TEST_FINISHED();
END_METHOD

METHOD PRIVATE Test_SINT
VAR
    a : SINT := 100;
    result : U_ExpectedOrActual;
END_VAR
TEST('Test_SINT');

result := TcUnit.F_AnyToUnionValue(AnyValue := a);

AssertEquals(Expected := a,
             Actual := result.sintExpectedOrActual,
             Message := 'Values differ');

TEST_FINISHED();
END_METHOD

METHOD PRIVATE Test_STRING
VAR
    a : STRING := 'This is a random string';
    result : U_ExpectedOrActual;
END_VAR
TEST('Test_STRING');

result := TcUnit.F_AnyToUnionValue(AnyValue := a);

AssertEquals(Expected := a,
             Actual := result.stringExpectedOrActual,
             Message := 'Values differ');

TEST_FINISHED();
END_METHOD

METHOD PRIVATE Test_STRING_2
VAR
    a : Tc2_System.T_MaxString := '8YNn5KOmPC4dAcpOBdLWnw4WkN126EwXsj65xeurG48gWBepinNaOIKeCVMtWNBSxQWPdtUYiAusDkjMLtQhDtiWbwvmoKcFwiUGDd7pOe0fd52J7hK60oaYAX6VWWmceLJX8utaDVrVzCGXafeZLeHl6jj5enfjg4tfb2WMEBdsBuG2iDKwzwhBLCPqXDnhe5HbemIbtZT7p62OEj2oDqiIYDD6tZdlhBCCelDBx6dbIp32wFm0TpRKsTiwkZ6'; // 255 characters
    result : U_ExpectedOrActual;
END_VAR
TEST('Test_STRING_2');

result := TcUnit.F_AnyToUnionValue(AnyValue := a);

AssertEquals(Expected := a,
             Actual := result.stringExpectedOrActual,
             Message := 'Values differ');

TEST_FINISHED();
END_METHOD

METHOD PRIVATE Test_TIME
VAR
    a : TIME := T#15M20S;
    result : U_ExpectedOrActual;
END_VAR
TEST('Test_TIME');

result := TcUnit.F_AnyToUnionValue(AnyValue := a);

AssertEquals(Expected := a,
             Actual := result.timeExpectedOrActual,
             Message := 'Values differ');

TEST_FINISHED();
END_METHOD

METHOD PRIVATE Test_TIME_OF_DAY
VAR
    a : TIME_OF_DAY := TOD#15:36:30.123;
    result : U_ExpectedOrActual;
END_VAR
TEST('Test_TIME_OF_DAY');

result := TcUnit.F_AnyToUnionValue(AnyValue := a);

AssertEquals(Expected := a,
             Actual := result.timeofdayExpectedOrActual,
             Message := 'Values differ');

TEST_FINISHED();
END_METHOD

METHOD PRIVATE Test_UDINT
VAR
    a : UDINT := 2555;
    result : U_ExpectedOrActual;
END_VAR
TEST('Test_UDINT');

result := TcUnit.F_AnyToUnionValue(AnyValue := a);

AssertEquals(Expected := a,
             Actual := result.udintExpectedOrActual,
             Message := 'Values differ');

TEST_FINISHED();
END_METHOD

METHOD PRIVATE Test_UINT
VAR
    a : UINT := 34523;
    result : U_ExpectedOrActual;
END_VAR
TEST('Test_UINT');

result := TcUnit.F_AnyToUnionValue(AnyValue := a);

AssertEquals(Expected := a,
             Actual := result.uintExpectedOrActual,
             Message := 'Values differ');

TEST_FINISHED();
END_METHOD

METHOD PRIVATE Test_ULINT
VAR
    a : ULINT := 25555423;
    result : U_ExpectedOrActual;
END_VAR
TEST('TEST_ULINT');

result := TcUnit.F_AnyToUnionValue(AnyValue := a);

AssertEquals(Expected := a,
             Actual := result.ulintExpectedOrActual,
             Message := 'Values differ');

TEST_FINISHED();
END_METHOD

METHOD PRIVATE Test_USINT
VAR
    a : USINT := 255;
    result : U_ExpectedOrActual;
END_VAR
TEST('Test_USINT');

result := TcUnit.F_AnyToUnionValue(AnyValue := a);

AssertEquals(Expected := a,
             Actual := result.usintExpectedOrActual,
             Message := 'Values differ');

TEST_FINISHED();
END_METHOD

METHOD PRIVATE Test_WORD
VAR
    a : WORD := 16#ABCD;
    result : U_ExpectedOrActual;
END_VAR
TEST('Test_WORD');

result := TcUnit.F_AnyToUnionValue(AnyValue := a);

AssertEquals(Expected := a,
             Actual := result.wordExpectedOrActual,
             Message := 'Values differ');

TEST_FINISHED();
END_METHOD

METHOD PRIVATE Test_WSTRING
VAR
    a : WSTRING := "This is a random string";
    result : U_ExpectedOrActual;
END_VAR
TEST('Test_WSTRING');

result := TcUnit.F_AnyToUnionValue(AnyValue := a);

AssertEquals(Expected := a,
             Actual := result.wstringExpectedOrActual,
             Message := 'Values differ');

TEST_FINISHED();
END_METHOD

END_FUNCTION_BLOCK

// ---- Test/FB_MultipleAssertWithSameParametersInSameCycleWithSameTest.TcPOU
(*
    This test-suite runs several asserts with the same parameters (same expected, actual, message) in the same cycle
    and in the same test.
    The reason we want the framework to support this is that theoretically the user could want to do an assert with the
    same message, in the same test, with the same data values for both expected and actual, although the data that the
    user does the assert on might be from different data sets.
*)
FUNCTION_BLOCK FB_MultipleAssertWithSameParametersInSameCycleWithSameTest EXTENDS TcUnit.FB_TestSuite

Assert_SeveralTimes();

METHOD PRIVATE Assert_SeveralTimes
VAR
    a : DWORD := 16#12345678;
    b : DWORD := 16#90ABCDEF;

    c : DWORD := 16#12345678;
    d : DWORD := 16#90ABCDEF;

    e : DWORD := 16#12345678;
    f : DWORD := 16#90ABCDEF;
END_VAR
TEST('Assert_SeveralTimes');

AssertEquals_DWORD(Expected := a,
                   Actual := b,
                   Message := 'Values differ');

AssertEquals_DWORD(Expected := c,
                   Actual := d,
                   Message := 'Values differ');

AssertEquals_DWORD(Expected := e,
                   Actual := f,
                   Message := 'Values differ');

TEST_FINISHED();
END_METHOD

END_FUNCTION_BLOCK

// ---- Test/FB_MultipleAssertWithSameParametersInDifferentCyclesButWithDifferentTests.TcPOU
(*
    This test-suite runs several asserts with the same parameters (same expected, actual, message), calling the asserts
    in different cycles and using different tests.
    On top of this, we will call new asserts (though with same parameters) in later cycles.
    The reason we want the framework to support this is that theoretically the user could want to do an assert with the
    same message, in different tests, with the same data values for both expected and actual, although the data that the
    user does the assert on might be from different data sets.
*)
{attribute 'call_after_init'}
FUNCTION_BLOCK FB_MultipleAssertWithSameParametersInDifferentCyclesButWithDifferentTests EXTENDS TcUnit.FB_TestSuite
VAR
    TimerAgain : Tc2_Standard.TON := (PT := T#1S); // Timer to call "AssertSeveralTimesAgain"
    TimerAgainAgain : Tc2_Standard.TON := (PT := T#5S); // Timer to call "AssertSeveralTimesAgainAgain"
    CalledAll : BOOL; // Indication of whether we've called all tests
END_VAR

TimerAgain(IN := TRUE);

Assert_SeveralTimes();

IF TimerAgain.Q THEN
    TimerAgainAgain(IN := TRUE);
    Assert_SeveralTimesAgain();
END_IF

IF TimerAgainAgain.Q THEN
    Assert_SeveralTimesAgainAgain();
    CalledAll := TRUE;
END_IF

METHOD PRIVATE Assert_SeveralTimes
VAR
    a : DWORD := 16#12345678;
    b : DWORD := 16#90ABCDEF;

    c : DWORD := 16#12345678;
    d : DWORD := 16#90ABCDEF;

    e : DWORD := 16#12345678;
    f : DWORD := 16#90ABCDEF;
END_VAR
TEST('Assert_SeveralTimes');

AssertEquals_DWORD(Expected := a,
                   Actual := b,
                   Message := 'Values differ');

AssertEquals_DWORD(Expected := c,
                   Actual := d,
                   Message := 'Values differ');

AssertEquals_DWORD(Expected := e,
                   Actual := f,
                   Message := 'Values differ');

IF CalledAll THEN
    TEST_FINISHED();
END_IF
END_METHOD

METHOD PRIVATE Assert_SeveralTimesAgain
VAR
    a : DWORD := 16#12345678;
    b : DWORD := 16#90ABCDEF;

    c : DWORD := 16#12345678;
    d : DWORD := 16#90ABCDEF;

    e : DWORD := 16#12345678;
    f : DWORD := 16#90ABCDEF;
END_VAR
TEST('Assert_SeveralTimesAgain');

AssertEquals_DWORD(Expected := a,
                   Actual := b,
                   Message := 'Values differ');

AssertEquals_DWORD(Expected := c,
                   Actual := d,
                   Message := 'Values differ');

AssertEquals_DWORD(Expected := e,
                   Actual := f,
                   Message := 'Values differ');

IF CalledAll THEN
    TEST_FINISHED();
END_IF
END_METHOD

METHOD PRIVATE Assert_SeveralTimesAgainAgain
VAR
    a : DWORD := 16#12345678;
    b : DWORD := 16#90ABCDEF;

    c : DWORD := 16#12345678;
    d : DWORD := 16#90ABCDEF;

    e : DWORD := 16#12345678;
    f : DWORD := 16#90ABCDEF;
END_VAR
TEST('Assert_SeveralTimesAgainAgain');

AssertEquals_DWORD(Expected := a,
                   Actual := b,
                   Message := 'Values differ');

AssertEquals_DWORD(Expected := c,
                   Actual := d,
                   Message := 'Values differ');

AssertEquals_DWORD(Expected := e,
                   Actual := f,
                   Message := 'Values differ');

IF CalledAll THEN
    TEST_FINISHED();
END_IF
END_METHOD

END_FUNCTION_BLOCK

// ---- Test/FB_MultipleAssertWithSameParametersInDifferentCyclesAndInSameTest.TcPOU
(*
    This test-suite runs several asserts with the same parameters (same expected, actual, message), calling the asserts
    in different cycles and using the same test.
    On top of this, we will call new asserts (though with same parameters) in later cycles.
    The reason we want the framework to support this is that theoretically the user could want to do an assert with the
    same message, using the same test with the same data values for both expected and actual, and splitting the asserts
    on different cycles.
*)
FUNCTION_BLOCK FB_MultipleAssertWithSameParametersInDifferentCyclesAndInSameTest EXTENDS TcUnit.FB_TestSuite
VAR
    TimerAgain : Tc2_Standard.TON := (PT := T#1S); // Timer to call "AssertSeveralTimesAgain"
    TimerAgainAgain : Tc2_Standard.TON := (PT := T#5S); // Timer to call "AssertSeveralTimesAgainAgain"
    CalledAll : BOOL; // Indication of whether we've called all tests
END_VAR

Assert_SeveralTimes();

METHOD PRIVATE Assert_SeveralTimes
VAR
    a : DWORD := 16#12345678;
    b : DWORD := 16#90ABCDEF;

    c : DWORD := 16#12345678;
    d : DWORD := 16#90ABCDEF;

    e : DWORD := 16#12345678;
    f : DWORD := 16#90ABCDEF;

    g : DWORD := 16#12345678;
    h : DWORD := 16#90ABCDEF;

    i : DWORD := 16#12345678;
    j : DWORD := 16#90ABCDEF;

    k : DWORD := 16#12345678;
    l : DWORD := 16#90ABCDEF;

    m : DWORD := 16#12345678;
    n : DWORD := 16#90ABCDEF;

    o : DWORD := 16#12345678;
    p : DWORD := 16#90ABCDEF;

    q : DWORD := 16#12345678;
    rr : DWORD := 16#90ABCDEF;
END_VAR
TEST('Assert_SeveralTimes');

AssertEquals_DWORD(Expected := a,
                   Actual := b,
                   Message := 'Values differ');
AssertEquals_DWORD(Expected := c,
                   Actual := d,
                   Message := 'Values differ');
AssertEquals_DWORD(Expected := e,
                   Actual := f,
                   Message := 'Values differ');

TimerAgain(IN := TRUE);
IF TimerAgain.Q THEN
    TimerAgainAgain(IN := TRUE);
    AssertEquals_DWORD(Expected := g,
                       Actual := h,
                       Message := 'Values differ');
    AssertEquals_DWORD(Expected := i,
                       Actual := j,
                       Message := 'Values differ');
    AssertEquals_DWORD(Expected := k,
                       Actual := l,
                       Message := 'Values differ');
END_IF

IF TimerAgainAgain.Q THEN
    AssertEquals_DWORD(Expected := m,
                       Actual := n,
                       Message := 'Values differ');
    AssertEquals_DWORD(Expected := o,
                       Actual := p,
                       Message := 'Values differ');
    AssertEquals_DWORD(Expected := q,
                       Actual := rr,
                       Message := 'Values differ');
    CalledAll := TRUE;
    TEST_FINISHED();
END_IF
END_METHOD

END_FUNCTION_BLOCK

// ---- Test/FB_SkipAssertionsWhenFinished.TcPOU
(*
    Contains tests that require multiple cycles:
    - A short test that finishes quickly
        - The assert statements all pass while the test is not finished
        - After the test is finished, the variables change so that the assert statements now fail,
            which shouldn't matter because the test is finished
    - A long test that finishes slowly
        - This test exists so that the entire test suite keeps running after the short test finishes
*)
FUNCTION_BLOCK FB_SkipAssertionsWhenFinished EXTENDS TcUnit.FB_TestSuite
VAR
    ShortTimer : Tc2_Standard.TON := (PT := T#200MS);
    LongTimer : Tc2_Standard.TON := (PT := T#1S);
END_VAR

Test_LongTest(ADR(LongTimer));
Test_ShortTest(ADR(ShortTimer));
Test_AssertImmediatelyAfterFinished();

(*
    Assertions called immediately after (and within the same cycle as) TEST_FINISHED should be
    ignored.
*)
METHOD Test_AssertImmediatelyAfterFinished
TEST('Test_AssertImmediatelyAfterFinished');
TEST_FINISHED();

AssertTrue(FALSE, 'This failing assertion should be skipped because the test is finished');
END_METHOD

METHOD Test_LongTest
VAR_INPUT
    Timer : POINTER TO Tc2_Standard.TON;
END_VAR
TEST('Test_LongTest');

Timer^(IN := TRUE);
IF Timer^.Q THEN
    TEST_FINISHED();
END_IF
END_METHOD

METHOD Test_ShortTest
VAR_INPUT
    Timer : POINTER TO Tc2_Standard.TON;
END_VAR
TEST('Test_ShortTest');

AssertFalse(Timer^.Q, 'This assertion will start to fail after the test is over, but it will be skipped at that point');

Timer^(IN := TRUE);
IF Timer^.Q THEN
    TEST_FINISHED();
END_IF
END_METHOD

END_FUNCTION_BLOCK

// ---- Test/FB_EmptyTestSuite.TcPOU
(* This is an empty testsuite with no test cases, so that we can verify that the system still prints the
   test results. *)
FUNCTION_BLOCK FB_EmptyTestSuite EXTENDS TcUnit.FB_TestSuite
VAR
END_VAR

END_FUNCTION_BLOCK

// ---- Test/FB_CheckIfSpecificTestIsFinished.TcPOU
(*
    Verifies that the function IS_TEST_FINISHED('Name') works as intended.
*)
FUNCTION_BLOCK FB_CheckIfSpecificTestIsFinished EXTENDS TcUnit.FB_TestSuite

CheckBeforeAndAfterFinishing();

METHOD CheckBeforeAndAfterFinishing
TEST('CheckBeforeAndAfterFinishing');

AssertEquals_BOOL(Expected := FALSE,
                  Actual := IS_TEST_FINISHED('CheckBeforeAndAfterFinishing'),
                  Message:='Values differ before finishing');

TEST_FINISHED();

AssertEquals_BOOL(Expected := TRUE,
                  Actual := IS_TEST_FINISHED('CheckBeforeAndAfterFinishing'),
                  Message:='Values differ after finishing');
END_METHOD

END_FUNCTION_BLOCK

// ---- Test/FB_WriteProtectedFunctions.TcPOU
(*
    This testsuite tests the WRITE_PROTECTED_* helper functions.
*)
FUNCTION_BLOCK FB_WriteProtectedFunctions EXTENDS TcUnit.FB_TestSuite

Test_WRITE_PROTECTED_BOOL();
Test_WRITE_PROTECTED_BYTE();
Test_WRITE_PROTECTED_DATE();
Test_WRITE_PROTECTED_DATE_AND_TIME();
Test_WRITE_PROTECTED_DINT();
Test_WRITE_PROTECTED_DWORD();
Test_WRITE_PROTECTED_INT();
Test_WRITE_PROTECTED_LREAL();
Test_WRITE_PROTECTED_REAL();
Test_WRITE_PROTECTED_SINT();
Test_WRITE_PROTECTED_STRING();
Test_WRITE_PROTECTED_TIME();
Test_WRITE_PROTECTED_TIME_OF_DAY();
Test_WRITE_PROTECTED_UDINT();
Test_WRITE_PROTECTED_UINT();
Test_WRITE_PROTECTED_USINT();
Test_WRITE_PROTECTED_WORD();

METHOD Test_WRITE_PROTECTED_BOOL
VAR
    ProtectedVariables : FB_ProtectedVariables;
END_VAR
TEST('Test_WRITE_PROTECTED_BOOL');

WRITE_PROTECTED_BOOL(ADR(ProtectedVariables.InputBOOL), TRUE);
AssertEquals_BOOL(TRUE, ProtectedVariables.InputBOOL, 'Overwriting protected InputBOOL');

WRITE_PROTECTED_BOOL(ADR(ProtectedVariables.VarBOOL), TRUE);
AssertEquals_BOOL(TRUE, ProtectedVariables.VarBOOL, 'Overwriting protected VarBOOL');

TEST_FINISHED();
END_METHOD

METHOD Test_WRITE_PROTECTED_BYTE
VAR
    ProtectedVariables : FB_ProtectedVariables;
END_VAR
TEST('Test_WRITE_PROTECTED_BYTE');

WRITE_PROTECTED_BYTE(ADR(ProtectedVariables.InputBYTE), 1);
AssertEquals_BYTE(1, ProtectedVariables.InputBYTE, 'Overwriting protected InputBYTE');

WRITE_PROTECTED_BYTE(ADR(ProtectedVariables.VarBYTE), 1);
AssertEquals_BYTE(1, ProtectedVariables.VarBYTE, 'Overwriting protected VarBYTE');

TEST_FINISHED();
END_METHOD

METHOD Test_WRITE_PROTECTED_DATE
VAR
    ProtectedVariables : FB_ProtectedVariables;
END_VAR
TEST('Test_WRITE_PROTECTED_DATE');

WRITE_PROTECTED_DATE(ADR(ProtectedVariables.InputDATE), D#2000-01-01);
AssertEquals_DATE(D#2000-01-01, ProtectedVariables.InputDATE, 'Overwriting protected InputDATE');

WRITE_PROTECTED_DATE(ADR(ProtectedVariables.VarDATE), D#2000-01-01);
AssertEquals_DATE(D#2000-01-01, ProtectedVariables.VarDATE, 'Overwriting protected VarDATE');

TEST_FINISHED();
END_METHOD

METHOD Test_WRITE_PROTECTED_DATE_AND_TIME
VAR
    ProtectedVariables : FB_ProtectedVariables;
END_VAR
TEST('Test_WRITE_PROTECTED_DATE_AND_TIME');

WRITE_PROTECTED_DATE_AND_TIME(ADR(ProtectedVariables.InputDATE_AND_TIME), DT#2000-01-01-00:00);
AssertEquals_DATE_AND_TIME(DT#2000-01-01-00:00, ProtectedVariables.InputDATE_AND_TIME, 'Overwriting protected InputDATE_AND_TIME');

WRITE_PROTECTED_DATE_AND_TIME(ADR(ProtectedVariables.VarDATE_AND_TIME), DT#2000-01-01-00:00);
AssertEquals_DATE_AND_TIME(DT#2000-01-01-00:00, ProtectedVariables.VarDATE_AND_TIME, 'Overwriting protected VarDATE_AND_TIME');

TEST_FINISHED();
END_METHOD

METHOD Test_WRITE_PROTECTED_DINT
VAR
    ProtectedVariables : FB_ProtectedVariables;
END_VAR
TEST('Test_WRITE_PROTECTED_DINT');

WRITE_PROTECTED_DINT(ADR(ProtectedVariables.InputDINT), 1);
AssertEquals_DINT(1, ProtectedVariables.InputDINT, 'Overwriting protected InputDINT');

WRITE_PROTECTED_DINT(ADR(ProtectedVariables.VarDINT), 1);
AssertEquals_DINT(1, ProtectedVariables.VarDINT, 'Overwriting protected VarDINT');

TEST_FINISHED();
END_METHOD

METHOD Test_WRITE_PROTECTED_DWORD
VAR
    ProtectedVariables : FB_ProtectedVariables;
END_VAR
TEST('Test_WRITE_PROTECTED_DWORD');

WRITE_PROTECTED_DWORD(ADR(ProtectedVariables.InputDWORD), 1);
AssertEquals_DWORD(1, ProtectedVariables.InputDWORD, 'Overwriting protected InputDWORD');

WRITE_PROTECTED_DWORD(ADR(ProtectedVariables.VarDWORD), 1);
AssertEquals_DWORD(1, ProtectedVariables.VarDWORD, 'Overwriting protected VarDWORD');

TEST_FINISHED();
END_METHOD

METHOD Test_WRITE_PROTECTED_INT
VAR
    ProtectedVariables : FB_ProtectedVariables;
END_VAR
TEST('Test_WRITE_PROTECTED_INT');

WRITE_PROTECTED_INT(ADR(ProtectedVariables.InputINT), 1);
AssertEquals_INT(1, ProtectedVariables.InputINT, 'Overwriting protected InputINT');

WRITE_PROTECTED_INT(ADR(ProtectedVariables.VarINT), 1);
AssertEquals_INT(1, ProtectedVariables.VarINT, 'Overwriting protected VarINT');

TEST_FINISHED();
END_METHOD

METHOD Test_WRITE_PROTECTED_LREAL
VAR
    ProtectedVariables : FB_ProtectedVariables;
END_VAR
TEST('Test_WRITE_PROTECTED_LREAL');

WRITE_PROTECTED_LREAL(ADR(ProtectedVariables.InputLREAL), 1);
AssertEquals_LREAL(1, ProtectedVariables.InputLREAL, 0, 'Overwriting protected InputLREAL');

WRITE_PROTECTED_LREAL(ADR(ProtectedVariables.VarLREAL), 1);
AssertEquals_LREAL(1, ProtectedVariables.VarLREAL, 0, 'Overwriting protected VarLREAL');

TEST_FINISHED();
END_METHOD

METHOD Test_WRITE_PROTECTED_REAL
VAR
    ProtectedVariables : FB_ProtectedVariables;
END_VAR
TEST('Test_WRITE_PROTECTED_REAL');

WRITE_PROTECTED_REAL(ADR(ProtectedVariables.InputREAL), 1);
AssertEquals_REAL(1, ProtectedVariables.InputREAL, 0, 'Overwriting protected InputREAL');

WRITE_PROTECTED_REAL(ADR(ProtectedVariables.VarREAL), 1);
AssertEquals_REAL(1, ProtectedVariables.VarREAL, 0, 'Overwriting protected VarREAL');

TEST_FINISHED();
END_METHOD

METHOD Test_WRITE_PROTECTED_SINT
VAR
    ProtectedVariables : FB_ProtectedVariables;
END_VAR
TEST('Test_WRITE_PROTECTED_SINT');

WRITE_PROTECTED_SINT(ADR(ProtectedVariables.InputSINT), 1);
AssertEquals_SINT(1, ProtectedVariables.InputSINT, 'Overwriting protected InputSINT');

WRITE_PROTECTED_SINT(ADR(ProtectedVariables.VarSINT), 1);
AssertEquals_SINT(1, ProtectedVariables.VarSINT, 'Overwriting protected VarSINT');

TEST_FINISHED();
END_METHOD

METHOD Test_WRITE_PROTECTED_STRING
VAR
    ProtectedVariables : FB_ProtectedVariables;
END_VAR
TEST('Test_WRITE_PROTECTED_STRING');

WRITE_PROTECTED_STRING(ADR(ProtectedVariables.InputSTRING), 'words');
AssertEquals_STRING('words', ProtectedVariables.InputSTRING, 'Overwriting protected InputSTRING');

WRITE_PROTECTED_STRING(ADR(ProtectedVariables.VarSTRING), 'words');
AssertEquals_STRING('words', ProtectedVariables.VarSTRING, 'Overwriting protected VarSTRING');

TEST_FINISHED();
END_METHOD

METHOD Test_WRITE_PROTECTED_TIME
VAR
    ProtectedVariables : FB_ProtectedVariables;
END_VAR
TEST('Test_WRITE_PROTECTED_TIME');

WRITE_PROTECTED_TIME(ADR(ProtectedVariables.InputTIME), T#1S);
AssertEquals_TIME(T#1S, ProtectedVariables.InputTIME, 'Overwriting protected InputTIME');

WRITE_PROTECTED_TIME(ADR(ProtectedVariables.VarTIME), T#1S);
AssertEquals_TIME(T#1S, ProtectedVariables.VarTIME, 'Overwriting protected VarTIME');

TEST_FINISHED();
END_METHOD

METHOD Test_WRITE_PROTECTED_TIME_OF_DAY
VAR
    ProtectedVariables : FB_ProtectedVariables;
END_VAR
TEST('Test_WRITE_PROTECTED_TIME_OF_DAY');

WRITE_PROTECTED_TIME_OF_DAY(ADR(ProtectedVariables.InputTIME_OF_DAY), TOD#11:11);
AssertEquals_TIME_OF_DAY(TOD#11:11, ProtectedVariables.InputTIME_OF_DAY, 'Overwriting protected InputTIME_OF_DAY');

WRITE_PROTECTED_TIME_OF_DAY(ADR(ProtectedVariables.VarTIME_OF_DAY), TOD#11:11);
AssertEquals_TIME_OF_DAY(TOD#11:11, ProtectedVariables.VarTIME_OF_DAY, 'Overwriting protected VarTIME_OF_DAY');

TEST_FINISHED();
END_METHOD

METHOD Test_WRITE_PROTECTED_UDINT
VAR
    ProtectedVariables : FB_ProtectedVariables;
END_VAR
TEST('Test_WRITE_PROTECTED_UDINT');

WRITE_PROTECTED_UDINT(ADR(ProtectedVariables.InputUDINT), 1);
AssertEquals_UDINT(1, ProtectedVariables.InputUDINT, 'Overwriting protected InputUDINT');

WRITE_PROTECTED_UDINT(ADR(ProtectedVariables.VarUDINT), 1);
AssertEquals_UDINT(1, ProtectedVariables.VarUDINT, 'Overwriting protected VarUDINT');

TEST_FINISHED();
END_METHOD

METHOD Test_WRITE_PROTECTED_UINT
VAR
    ProtectedVariables : FB_ProtectedVariables;
END_VAR
TEST('Test_WRITE_PROTECTED_UINT');

WRITE_PROTECTED_UINT(ADR(ProtectedVariables.InputUINT), 1);
AssertEquals_UINT(1, ProtectedVariables.InputUINT, 'Overwriting protected InputUINT');

WRITE_PROTECTED_UINT(ADR(ProtectedVariables.VarUINT), 1);
AssertEquals_UINT(1, ProtectedVariables.VarUINT, 'Overwriting protected VarUINT');

TEST_FINISHED();
END_METHOD

METHOD Test_WRITE_PROTECTED_USINT
VAR
    ProtectedVariables : FB_ProtectedVariables;
END_VAR
TEST('Test_WRITE_PROTECTED_USINT');

WRITE_PROTECTED_USINT(ADR(ProtectedVariables.InputUSINT), 1);
AssertEquals_USINT(1, ProtectedVariables.InputUSINT, 'Overwriting protected InputUSINT');

WRITE_PROTECTED_USINT(ADR(ProtectedVariables.VarUSINT), 1);
AssertEquals_USINT(1, ProtectedVariables.VarUSINT, 'Overwriting protected VarUSINT');

TEST_FINISHED();
END_METHOD

METHOD Test_WRITE_PROTECTED_WORD
VAR
    ProtectedVariables : FB_ProtectedVariables;
END_VAR
TEST('Test_WRITE_PROTECTED_WORD');

WRITE_PROTECTED_WORD(ADR(ProtectedVariables.InputWORD), 1);
AssertEquals_WORD(1, ProtectedVariables.InputWORD, 'Overwriting protected InputWORD');

WRITE_PROTECTED_WORD(ADR(ProtectedVariables.VarWORD), 1);
AssertEquals_WORD(1, ProtectedVariables.VarWORD, 'Overwriting protected VarWORD');

TEST_FINISHED();
END_METHOD

END_FUNCTION_BLOCK

// ---- POUs/FB_ProtectedVariables.TcPOU
(*
    Contains different types of "protected" variables that you could not normally write to in
    production PLC code, but would need to overwrite for testing purposes. Used for testing the
    WRITE_PROTECTED_* functions, but this FB doesn't contain any tests itself.
*)
FUNCTION_BLOCK FB_ProtectedVariables
VAR_INPUT
    InputBOOL AT %I* : BOOL;
    InputBYTE AT %I* : BYTE;
    InputDATE AT %I* : DATE;
    InputDATE_AND_TIME AT %I* : DATE_AND_TIME;
    InputDINT AT %I* : DINT;
    InputDWORD AT %I* : DWORD;
    InputINT AT %I* : INT;
    InputLREAL AT %I* : LREAL;
    InputREAL AT %I* : REAL;
    InputSINT AT %I* : SINT;
    InputSTRING AT %I* : STRING;
    InputTIME AT %I* : TIME;
    InputTIME_OF_DAY AT %I* : TIME_OF_DAY;
    InputUDINT AT %I* : UDINT;
    InputUINT AT %I* : UINT;
    InputUSINT AT %I* : USINT;
    InputWORD AT %I* : WORD;
END_VAR
VAR
    VarBOOL : BOOL;
    VarBYTE : BYTE;
    VarDATE : DATE;
    VarDATE_AND_TIME : DATE_AND_TIME;
    VarDINT : DINT;
    VarDWORD : DWORD;
    VarINT : INT;
    VarLREAL : LREAL;
    VarREAL : REAL;
    VarSINT : SINT;
    VarSTRING : STRING;
    VarTIME : TIME;
    VarTIME_OF_DAY : TIME_OF_DAY;
    VarUDINT : UDINT;
    VarUINT : UINT;
    VarUSINT : USINT;
    VarWORD : WORD;
END_VAR

END_FUNCTION_BLOCK

// ---- Test/FB_TestFinishedNamed.TcPOU
(* This function blocks tests the TEST_FINISHED_NAMED function by creating various tests
   and finishing them in steps *)
FUNCTION_BLOCK FB_TestFinishedNamed EXTENDS TcUnit.FB_TestSuite
VAR
    
END_VAR

END_FUNCTION_BLOCK

// ---- Test/FB_AdjustAssertFailureMessageToMax253CharLengthTest.TcPOU
(* This testsuite tests the function block FB_AdjustAssertFailureMessageToMax255CharLength_Test
   The total printed message can not be more than 253 characters long.
*)
FUNCTION_BLOCK FB_AdjustAssertFailureMessageToMax253CharLengthTest EXTENDS TcUnit.FB_TestSuite

TestInstancePath253CharsExpectTooLongTestInstancePath();
TestInstancePath221CharsExpectShortenedTestInstancePath();
TestInstancePath255CharsExpectTooLongTestInstancePath();

METHOD TestInstancePath221CharsExpectShortenedTestInstancePath
VAR
    AdjustAssertFailureMessageToMax253CharLength : FB_AdjustAssertFailureMessageToMax253CharLength;

    // @Text-Fixture
    TestInstancePathNameWith221Chars : Tc2_System.T_MaxString := 'PRG_TEST.LongInstanceNameLongInstanceNameLongInstanceNameLongInstanceNameLongInstanceNameLongInstanceNameLongInstanceNameLongInstanceNameLongInstanceNameLongInstanceName@LONGTESTNAMELONGTESTNAMELONGTESTNAMELONGTESTNAMELON';
    TooLongTestMessage60Chars : Tc2_System.T_MaxString := 'Very long message that is 60 characters long which means tha';
    
    // @Test-Result-Expected
    // 221 + 32 = 253 (in other words, expected test message should be 32 characters long including '...TestMsg too long'
    TestMessageResultExpected : Tc2_System.T_MaxString := 'Very long mes...TestMsg too long'; 

    // @Test-Result
    TestInstancePathResult : Tc2_System.T_MaxString;
    TestMessageResult : Tc2_System.T_MaxString;
END_VAR
TEST('TestInstancePath221CharsExpectShortenedTestInstancePath');

AdjustAssertFailureMessageToMax253CharLength(MsgFmtString := TestInstancePathNameWith221Chars,
                                             StringArg := TooLongTestMessage60Chars,
                                             MsgFmtStringProcessed => TestInstancePathResult,
                                             StringArgProcessed => TestMessageResult);


AssertEquals_STRING(Expected := TestInstancePathNameWith221Chars, // Same test instance path should be expected as the one going in
                    Actual := TestInstancePathResult,
                    'Test instance path not correct');

AssertEquals_STRING(Expected := TestMessageResultExpected,
                    Actual := TestMessageResult,
                    'Test message not correct');

TEST_FINISHED();
END_METHOD

METHOD PRIVATE TestInstancePath253CharsExpectTooLongTestInstancePath
VAR
    AdjustAssertFailureMessageToMax253CharLength : FB_AdjustAssertFailureMessageToMax253CharLength;

    // @Text-Fixture
    TestInstancePathNameWith253Chars : Tc2_System.T_MaxString := 'PRG_TEST.LongInstanceNameLongInstanceNameLongInstanceNameLongInstanceNameLongInstanceNameLongInstanceNameLongInstanceNameLongInstanceNameLongInstanceNameLongInstanceName@LONGTESTNAMELONGTESTNAMELONGTESTNAMELONGTESTNAMELONGTESTNAMELONGTESTNAMELONGTESTNAM';
    ShortTestMessage : Tc2_System.T_MaxString := 'Very short message';

    // @Test-Result-Expected
    TestInstancePathNameWith253CharsExpectedResult : Tc2_System.T_MaxString := 'PRG_TEST.LongInstanceNameLongInstanceNameLongInstanceNameLongInstanceNameLongInstanceNameLongInstanceNameLongInstanceNameLongInstanceNameLongInstanceNameLongInstanceName@LONGTESTNAMELONGTESTNAMELONGTESTNAMELONGTESTNAMELONGTESTNAMELON...TestName too long';
    ShortTestMessageExpectedResult : Tc2_System.T_MaxString := '';

    // @Test-Result
    TestInstancePathNameWith253CharsResult : Tc2_System.T_MaxString;
    ShortTestMessageResult : Tc2_System.T_MaxString;
END_VAR
TEST('TestInstancePath253CharsExpectTooLongTestInstancePath');

AdjustAssertFailureMessageToMax253CharLength(MsgFmtString := TestInstancePathNameWith253Chars,
                                             StringArg := ShortTestMessage,
                                             MsgFmtStringProcessed => TestInstancePathNameWith253CharsResult,
                                             StringArgProcessed => ShortTestMessageResult);

AssertEquals_STRING(Expected := TestInstancePathNameWith253CharsExpectedResult,
                    Actual := TestInstancePathNameWith253CharsResult,
                    'Test instance path not correct');

AssertEquals_STRING(Expected := ShortTestMessageExpectedResult,
                    Actual := ShortTestMessageResult,
                    'Test message not correct');

TEST_FINISHED();
END_METHOD

METHOD PRIVATE TestInstancePath255CharsExpectTooLongTestInstancePath
VAR
    AdjustAssertFailureMessageToMax253CharLength : FB_AdjustAssertFailureMessageToMax253CharLength;

    // @Text-Fixture
    TestInstancePathNameWith255Chars : Tc2_System.T_MaxString := 'PRG_TEST.LongInstanceNameLongInstanceNameLongInstanceNameLongInstanceNameLongInstanceNameLongInstanceNameLongInstanceNameLongInstanceNameLongInstanceNameLongInstanceName@LONGTESTNAMELONGTESTNAMELONGTESTNAMELONGTESTNAMELONGTESTNAMELONGTESTNAMELONGTESTNAGAV';
    ShortTestMessage : Tc2_System.T_MaxString := 'Very short message';

    // @Test-Result-Expected
    TestInstancePathNameWith253CharsExpectedResult : Tc2_System.T_MaxString := 'PRG_TEST.LongInstanceNameLongInstanceNameLongInstanceNameLongInstanceNameLongInstanceNameLongInstanceNameLongInstanceNameLongInstanceNameLongInstanceNameLongInstanceName@LONGTESTNAMELONGTESTNAMELONGTESTNAMELONGTESTNAMELONGTESTNAMELON...TestName too long';
    ShortTestMessageExpectedResult : Tc2_System.T_MaxString := '';

    // @Test-Result
    TestInstancePathNameWith253CharsResult : Tc2_System.T_MaxString;
    ShortTestMessageResult : Tc2_System.T_MaxString;
END_VAR
TEST('TestInstancePath255CharsExpectTooLongTestInstancePath');

AdjustAssertFailureMessageToMax253CharLength(MsgFmtString := TestInstancePathNameWith255Chars,
                                             StringArg := ShortTestMessage,
                                             MsgFmtStringProcessed => TestInstancePathNameWith253CharsResult,
                                             StringArgProcessed => ShortTestMessageResult);

AssertEquals_STRING(Expected := TestInstancePathNameWith253CharsExpectedResult,
                    Actual := TestInstancePathNameWith253CharsResult,
                    'Test instance path not correct');

AssertEquals_STRING(Expected := ShortTestMessageExpectedResult,
                    Actual := ShortTestMessageResult,
                    'Test message not correct');

TEST_FINISHED();
END_METHOD

END_FUNCTION_BLOCK

// ---- Test/FB_TestFinishedNamedDoesNotExist.TcPOU
(*
    This FB tests the free function TEST_FINISHED_NAMED. Calling this function with a name that doesn't exist should
    produce an error message that says so. This error message should also only be printed once.
*)
FUNCTION_BLOCK FB_TestFinishedNamedDoesNotExist EXTENDS TcUnit.FB_TestSuite
VAR
END_VAR

Test_FinishedNamed();

METHOD PRIVATE Test_FinishedNamed
VAR
    a : INT := 2;
    b : INT := 2;
    
    bajs : BOOL;
END_VAR
TEST('Test_FinishedNamed');

AssertEquals_INT(Expected := a,
                 Actual := b,
                 Message := 'Values differ');

TEST_FINISHED_NAMED('AnotherTestNameThatDoesNotExist');
END_METHOD

END_FUNCTION_BLOCK
